{attribute addProperty BoxType "EL1804-0000-0016"}
{attribute addProperty Id "ChannelAT %I*ARRAY[0..3] OF Channel_E4AEF59E3240WcStateAT %I*WcState_F855686C1620InfoDataAT %I*InfoData_192954DE1620"}
{attribute addProperty CRC "2345458285"}
{attribute addProperty SizeInBites "64"}
{attribute addProperty SizeInBytes "8"}
TYPE EL1804_5A15FBDA :
STRUCT
	{attribute addProperty Name "Channel"}
	Channel : ARRAY[0..3] OF Channel_E4AEF59E;
	{attribute addProperty Name "WcState"}
	WcState : WcState_F855686C;
	{attribute addProperty Name "InfoData"}
	InfoData : InfoData_192954DE;
END_STRUCT
END_TYPE

(* stored: Version 1.2.0.0, ProductVersion 3.1.4024.9
   DUT EL1804_5A15FBDA: Id {7dba0a05-b640-4f2c-b042-1a4bf4800e15} *)
